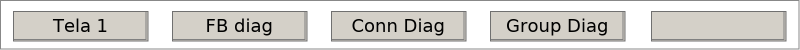
VISUALIZATION footer  // 800x50
    Button (13,11 135x30), "Tela 1"
        OnMouseClick: change screen: Visualization
    Button (172,11 135x30), "FB diag"
        OnMouseClick: change screen: FB_Diag
    Button (331,11 135x30), "Conn Diag"
        OnMouseClick: change screen: ConnDiag
    Button (490,11 135x30), "Group Diag"
        OnMouseClick: change screen: Group
    Button (651,11 135x30)
END_VISUALIZATION

(* stored: Version 1.1.0.1, ProductVersion 3.1.4024.12
   Visu footer: Id {ed4ef701-b1f6-491f-a520-0294465731b1} *)
